PROGRAM MAIN
VAR
END_VAR

END_PROGRAM

(* stored: Version 1.1.0.1
   POU MAIN: Id {6d485f51-279d-401b-9c8f-336fb57a731a} *)
